Fanuc KAREL source: ko00106.KL

PROGRAM KO00106
%STACKSIZE=65535
%PRIORITY=65535
%NOLOCKGROUP
VAR
A : REAL
B : INTEGER
OUT : REAL
BEGIN
A=1
B=2
-- UNRESOLVED_PC line 10 opcodes [27 22 27 21 64 76 23] marker_code=29
END KO00106
